# EPICS substitutions: testioApp/Db/output.substitutions
file ../../db/output.db {
    pattern	{Sys,	  	Pin, 	Logic, 	Desc}
		{"BBB01",	"60",	"H",	"Out 60 BeagleBone"}
#		{"BBB01", 	"56",	"H"	""}
}
